FUNCTION addVec7 : vec7d
VAR_IN_OUT CONSTANT
	i_vec1 :Vec7d;
	i_vec2 :Vec7d;
END_VAR
VAR
	i: INT ;
END_VAR

FOR i:=1 TO 7 DO 
	addVec7[i]:=i_vec1[i]+i_vec2[i];
END_FOR

END_FUNCTION

(* stored: Version 1.1.0.1, ProductVersion 3.1.4024.12
   POU addVec7: Id {7f08a62c-564e-4a4d-aa2c-e8ed8f70fa3e}, SpecialFunc None *)
